TYPE "UDT_Valve_ALM"
VERSION : 0.1
   STRUCT
      OUT_wALM : Word;   //  报警字 (Bit0=开阀超时报警, Bit1=关阀超时报警, Bit2=传感器故障报警)
      OUT_xSensorFault : Bool;   //  传感器故障
      OUT_xOpenTimeout : Bool;   //  开阀超时
      OUT_xCloseTimeout : Bool;   //  关阀超时
   END_STRUCT;

END_TYPE
